FUNCTION GetUsedStringLength : UDINT
VAR_INPUT
	pByte : POINTER TO BYTE; //use ADR(myString)
END_VAR
VAR
    i : UDINT := 0;
END_VAR

//every string in twincat is 0 terminated
IF pByte = 0 THEN
	RETURN;
END_IF

WHILE (pByte^ <> 0) DO
    pByte := pByte + 1; // Pointer auf das nächste Byte verschieben
    i := i + 1;
END_WHILE;

GetUsedStringLength := i;

END_FUNCTION

(* stored: Version 1.1.0.1, ProductVersion 3.1.4024.13
   POU GetUsedStringLength: Id {68254f53-56ca-44a3-98c9-c7dc875b6182}, SpecialFunc None *)
